ABB RobotStudio station: Solution progress.rsstn

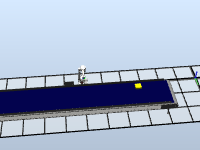
Station Solution1 (saved by RobotStudio 6.8.8148.134)
Controller System1, task T_ROB1: task frame (RAPID world) sits at (6016.55, 235.44, 350) mm, rotated rx 0 ry 0 rz 90 deg in the station
Controller System1
  mechanical unit ROB_1: IRB1600_10_145__01, 6 joints, base frame (0, 0, 0) mm
  mechanical unit CNV1: ?, 1 joints, base frame (0, 0, 0) mm
Layout (positions relative to the parent item):
  - bin mover_3 [smart component, from libraries\bin mover.rslib] at (-500, 0, 0) mm
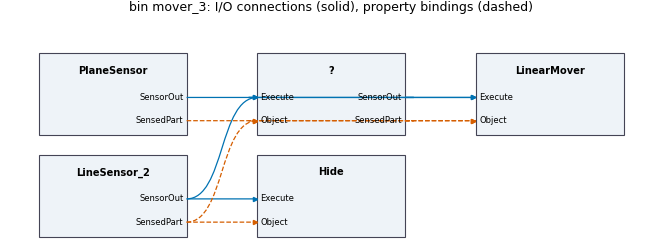
      connections:
        ?.SensorOut -> LinearMover.Execute
        PlaneSensor.SensorOut -> LinearMover.Execute
        ?.SensorOut -> ?.Execute
        LineSensor_2.SensorOut -> ?.Execute
        LineSensor_2.SensorOut -> Hide.Execute
        ?.SensedPart => LinearMover.Object
        PlaneSensor.SensedPart => LinearMover.Object
        ?.SensedPart => ?.Object
        LineSensor_2.SensedPart => ?.Object
        LineSensor_2.SensedPart => Hide.Object
    - LinearMover [smart component, from Components\LinearMover.rslib] at (6663.26, 677.27, 1050.93) mm, rotated rx 180 ry 0 rz 90 deg
        properties: Object=(none); Direction=[0 0 -1]; Speed=8; Reference=Global; ReferenceObject=(none)
    - PlaneSensor [smart component, from Components\PlaneSensor.rslib]
        properties: Origin=[7.419145 0.146999 1.42]; Axis1=[0 0 -1.35]; Axis2=[0 0.4 0]; SensedPart=(none)
      - _sensorPart_ [part, from libraries\bin mover.rslib]
    - LineSensor_2 [smart component, from Components\LineSensor.rslib]
        properties: Start=[7.369145 0.346999 0.008]; End=[7.369145 0.346999 0.123]; Radius=0.09; SensedPart=(none); SensedPoint=[0 0 0]
      - _sensorPart_ [part, from libraries\bin mover.rslib]
    - Hide [smart component, from Components\Hide.rslib]
        properties: Object=(none)
  - bin1_2 [part, from libraries\bin1.rslib] at (6733.74, 347, -12) mm
  - conveyor 1 [part] at (0, -1500, -4460) mm, rotated rx 90 ry 0 rz 90 deg
  - Suction gripper 18cm [smart component] at (6016.55, 985.44, 1386.5) mm, rotated rx 180 ry 0 rz -90 deg
      signals: DI do1
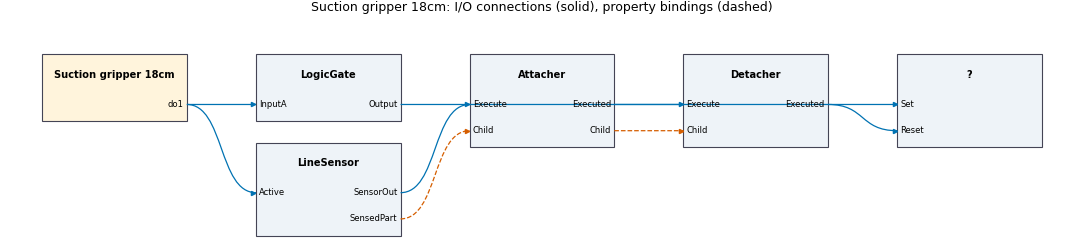
      connections:
        Suction gripper 18cm.do1 -> LogicGate.InputA
        Suction gripper 18cm.do1 -> LineSensor.Active
        LogicGate.Output -> Detacher.Execute
        LineSensor.SensorOut -> Attacher.Execute
        Attacher.Executed -> ?.Set
        Detacher.Executed -> ?.Reset
        LineSensor.SensedPart => Attacher.Child
        Attacher.Child => Detacher.Child
    - Attacher [smart component, from Components\Attacher.rslib]
        properties: Parent=(none); Flange=0; Child=(none); Mount=false; Offset=[0 0 0]; Orientation=[0 0 0]
    - LogicGate [smart component, from Components\LogicGate.rslib]
        properties: Operator=NOT; Delay=0
    - LineSensor [smart component, from Components\LineSensor.rslib] at (7150.29, 306.47, 1168.39) mm, rotated rx 180 ry 0 rz 90 deg
        properties: Start=[-0.30577796087058 -7.14894421240012 1.16938863540814]; End=[-0.305777964813962 -7.14894420825673 1.13938863540814]; Radius=0.09; SensedPart=(none); SensedPoint=[0 0 0]
      - _sensorPart_ [part]
    - Detacher [smart component, from Components\Detacher.rslib]
        properties: Child=(none); KeepPosition=true
  - Suction_gripper 18cm [mechanism, from libraries\Suction_gripper_18cm.rslib] at (6016.55, 985.44, 1471.5) mm, rotated rx 180 ry 0 rz -90 deg
  - IRB1600_10_145__01 [mechanism, from Robots\IRB1600_10_145_G_01.rslib] at (6016.55, 235.44, 350) mm, rotated rx 0 ry 0 rz 90 deg; joint values [0, 0, 0, 0, 1.5708, 0] (rad or m)
  - 输送链 [conveyor]
    - Conveyor cover [part] at (-300, 0, 14) mm
    - Yellow block [part] at (0, -475.41, 0) mm
    - 传送带对象_4 [conveyorobject] at (1835.63, 748.67, 709.58) mm
      - Yellow block [part] at (-1500, -1095, -698) mm
Attachment: Suction gripper 18cm is attached to Suction_gripper 18cm / Suction gripper 18cm
Attachment: Suction_gripper 18cm is attached to IRB1600_10_145__01 / Link6
Targets, tools, work objects and paths stored in the station, written as RAPID:
! task T_ROB1
MODULE CalibData
  PERS tooldata Suction_gripper_18cm:=[TRUE,[[0,0,85],[1,0,0,0]],[1,[0,0,1],[1,0,0,0],0,0,0]];
ENDMODULE

